// TIA Portal V17 export
// export: Created 2025-06-26T06:49:10.750176Z, ExportSetting WithDefaults, DisplayName Totally Integrated Automation Portal, DisplayVersion V17 Update 8, DisplayName TIA Portal Openness, DisplayVersion V17 Update 8, DisplayName TIA Portal Version Control Interface, DisplayVersion V17, DisplayName STEP 7 Professional, DisplayVersion V17 Update 8, DisplayName STEP 7 Safety, DisplayVersion V17 Update 6, DisplayName WinCC Advanced, DisplayVersion V17 Update 8
FUNCTION_BLOCK "DigitalInputProcessing"   // FB8, FBD
TITLE = Handle digital input signals
{ S7_Optimized_Access := 'TRUE' }
AUTHOR : Heaten
VERSION : 0.1
// Map, validate and process digital inputs
// stored: AutoNumber true, IsIECCheckEnabled false, IsRetainMemResEnabled false, MemoryReserve 0, SetENOAutomatically false, UDAEnableTagReadback false
   VAR
      HBL_LS_632 { ExternalAccessible := 'False'; ExternalVisible := 'False'; ExternalWritable := 'False'} : "stAnalogInput";
      HBL_LS_633 { S7_SetPoint := 'True'} : "stAnalogInput";
      HBL_LS_644 { S7_SetPoint := 'True'} : "stAnalogInput";
      HBL_LS_674 { S7_SetPoint := 'True'} : "stAnalogInput";
      Dummy { ExternalAccessible := 'False'; ExternalVisible := 'False'; ExternalWritable := 'False'} : Bool;
      LS632 : Real;
      LS633 : Real;
      LS644 : Real;
      LS674 : Real;
   END_VAR
   // HBL_LS_632.Raw.iMin := 0;
   // HBL_LS_632.Raw.iMax := 27648;
   // HBL_LS_632.Eng.fMin := 4.0;   // [mA]
   // HBL_LS_632.Eng.fMax := 20.0;   // [mA]
   // HBL_LS_633.Raw.iMin := 0;
   // HBL_LS_633.Raw.iMax := 27648;
   // HBL_LS_633.Eng.fMin := 4.0;   // [mA]
   // HBL_LS_633.Eng.fMax := 20.0;   // [mA]
   // HBL_LS_644.Eng.fMin := 4.0;
   // HBL_LS_644.Eng.fMax := 20.0;
   // HBL_LS_674.Eng.fMin := 4.0;
   // HBL_LS_674.Eng.fMax := 20.0;
BEGIN

REGION Network 1: Emergency stop status
   // Polarity of input is preserved. 1 = No E-stop, 0 = E-stop
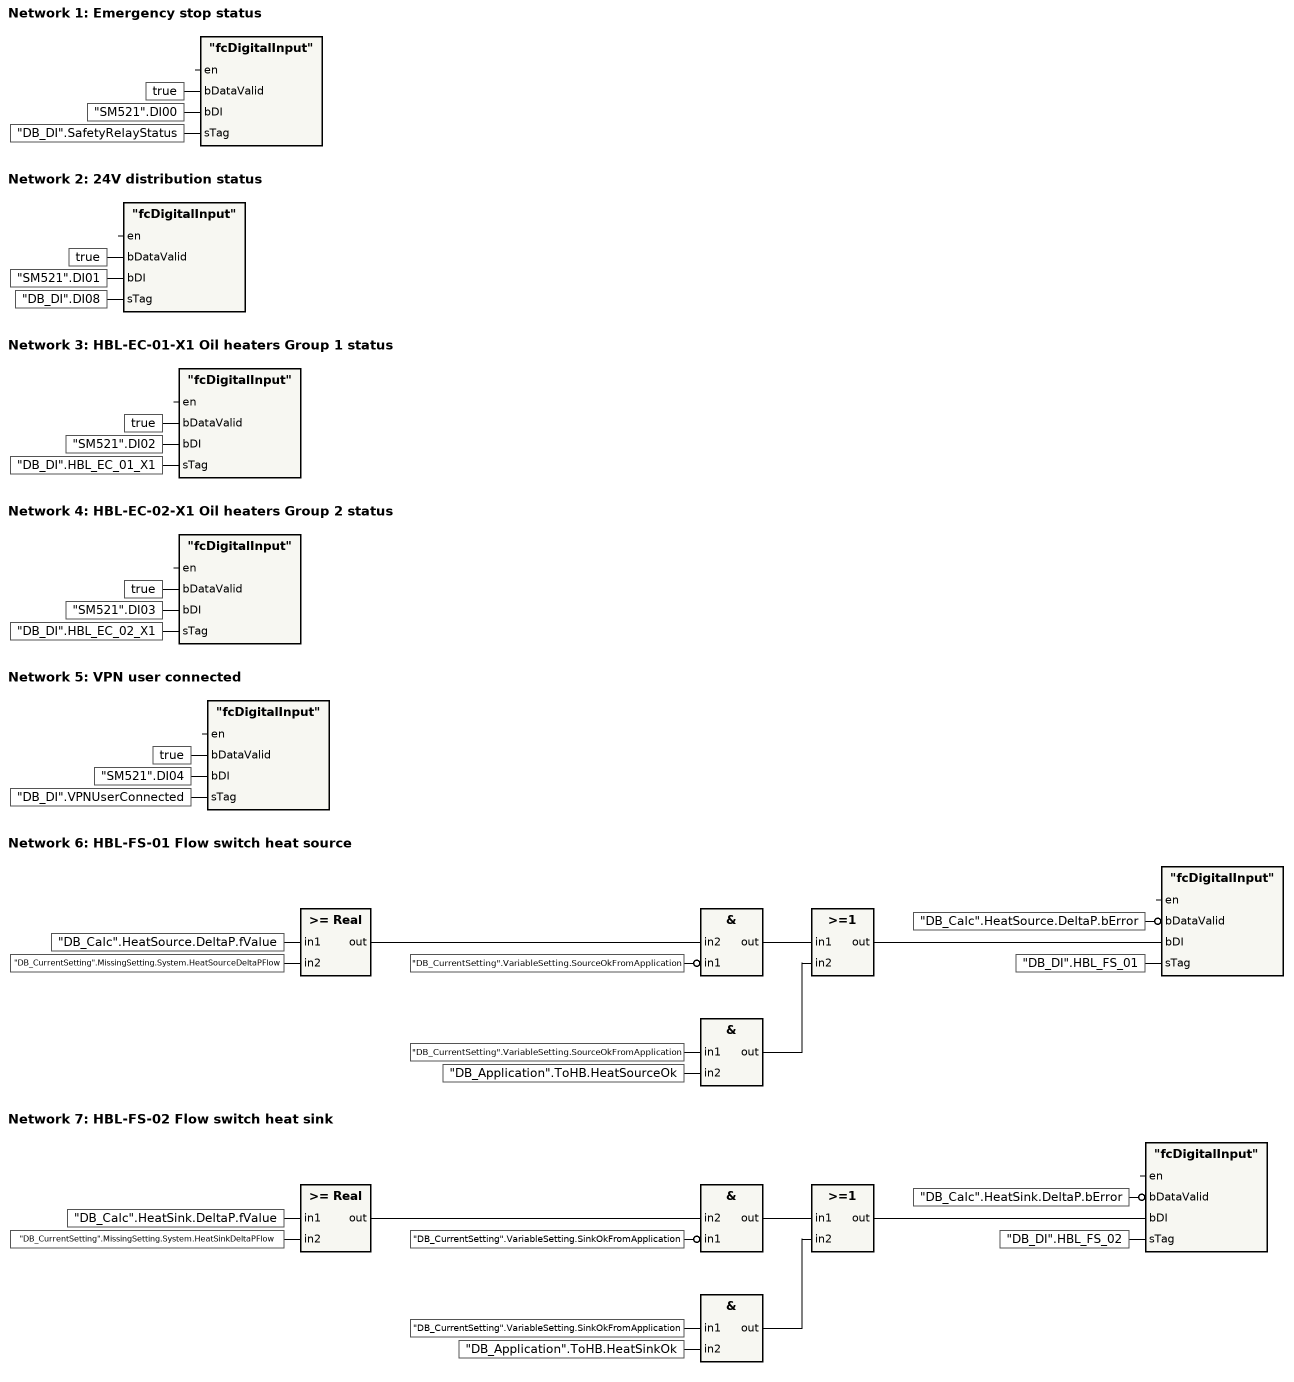
   "fcDigitalInput"(bDataValid := true, bDI := "SM521".DI00, sTag := "DB_DI".SafetyRelayStatus);
END_REGION

REGION Network 2: 24V distribution status
   "fcDigitalInput"(bDataValid := true, bDI := "SM521".DI01, sTag := "DB_DI".DI08);
END_REGION

REGION Network 3: HBL-EC-01-X1 Oil heaters Group 1 status
   "fcDigitalInput"(bDataValid := true, bDI := "SM521".DI02, sTag := "DB_DI".HBL_EC_01_X1);
END_REGION

REGION Network 4: HBL-EC-02-X1 Oil heaters Group 2 status
   "fcDigitalInput"(bDataValid := true, bDI := "SM521".DI03, sTag := "DB_DI".HBL_EC_02_X1);
END_REGION

REGION Network 5: VPN user connected
   "fcDigitalInput"(bDataValid := true, bDI := "SM521".DI04, sTag := "DB_DI".VPNUserConnected);
END_REGION

REGION Network 6: HBL-FS-01 Flow switch heat source
   // Virtual instrument:
   //  - Generate this locally from the pressure difference across the evaporator
   //  - Let the Application PLC do it based on input from the host process
   "fcDigitalInput"(bDataValid := NOT "DB_Calc".HeatSource.DeltaP.bError,
                    bDI := (("DB_Calc".HeatSource.DeltaP.fValue >= "DB_CurrentSetting".MissingSetting.System.HeatSourceDeltaPFlow) AND NOT "DB_CurrentSetting".VariableSetting.SourceOkFromApplication) OR ("DB_CurrentSetting".VariableSetting.SourceOkFromApplication AND "DB_Application".ToHB.HeatSourceOk),
                    sTag := "DB_DI".HBL_FS_01);
END_REGION

REGION Network 7: HBL-FS-02 Flow switch heat sink
   // Virtual instrument:
   //  - Generate this from the pressure difference across the condenser
   //  - Let the Application PLC does it based on input from the host process
   "fcDigitalInput"(bDataValid := NOT "DB_Calc".HeatSink.DeltaP.bError,
                    bDI := (("DB_Calc".HeatSink.DeltaP.fValue >= "DB_CurrentSetting".MissingSetting.System.HeatSinkDeltaPFlow) AND NOT "DB_CurrentSetting".VariableSetting.SinkOkFromApplication) OR ("DB_CurrentSetting".VariableSetting.SinkOkFromApplication AND "DB_Application".ToHB.HeatSinkOk),
                    sTag := "DB_DI".HBL_FS_02);
END_REGION

REGION Network 8: HBL-PS-500-X2 Compressor discharge overpressure
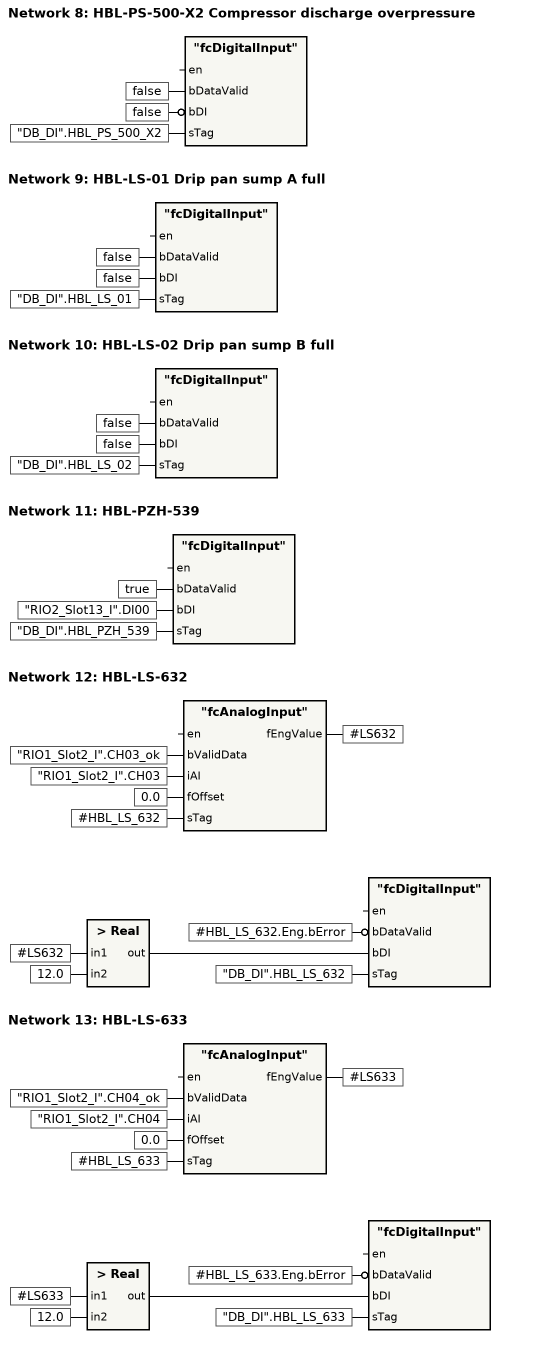
   "fcDigitalInput"(bDataValid := false, bDI := NOT false, sTag := "DB_DI".HBL_PS_500_X2);
END_REGION

REGION Network 9: HBL-LS-01 Drip pan sump A full
   "fcDigitalInput"(bDataValid := false, bDI := false, sTag := "DB_DI".HBL_LS_01);
END_REGION

REGION Network 10: HBL-LS-02 Drip pan sump B full
   "fcDigitalInput"(bDataValid := false, bDI := false, sTag := "DB_DI".HBL_LS_02);
END_REGION

REGION Network 11: HBL-PZH-539
   "fcDigitalInput"(bDataValid := true, bDI := "RIO2_Slot13_I".DI00, sTag := "DB_DI".HBL_PZH_539);
END_REGION

REGION Network 12: HBL-LS-632
   // 2-wire level switch. Low = 8mA, High = 16mA. Use a 12mA threshold to switch HI/LO
   "fcAnalogInput"(bValidData := "RIO1_Slot2_I".CH03_ok,
                   iAI := "RIO1_Slot2_I".CH03,
                   fOffset := 0.0,
                   sTag := #HBL_LS_632,
                   fEngValue => #LS632);
   "fcDigitalInput"(bDataValid := NOT #HBL_LS_632.Eng.bError, bDI := #LS632 > 12.0, sTag := "DB_DI".HBL_LS_632);
END_REGION

REGION Network 13: HBL-LS-633
   // 2-wire level switch. Low = 8mA, High = 16mA. Use a 12mA threshold to switch HI/LO
   "fcAnalogInput"(bValidData := "RIO1_Slot2_I".CH04_ok,
                   iAI := "RIO1_Slot2_I".CH04,
                   fOffset := 0.0,
                   sTag := #HBL_LS_633,
                   fEngValue => #LS633);
   "fcDigitalInput"(bDataValid := NOT #HBL_LS_633.Eng.bError, bDI := #LS633 > 12.0, sTag := "DB_DI".HBL_LS_633);
END_REGION

REGION Network 14: HBL-LS-644
   // 2-wire level switch. Low = 8mA, High = 16mA. Use a 12mA threshold to switch HI/LO
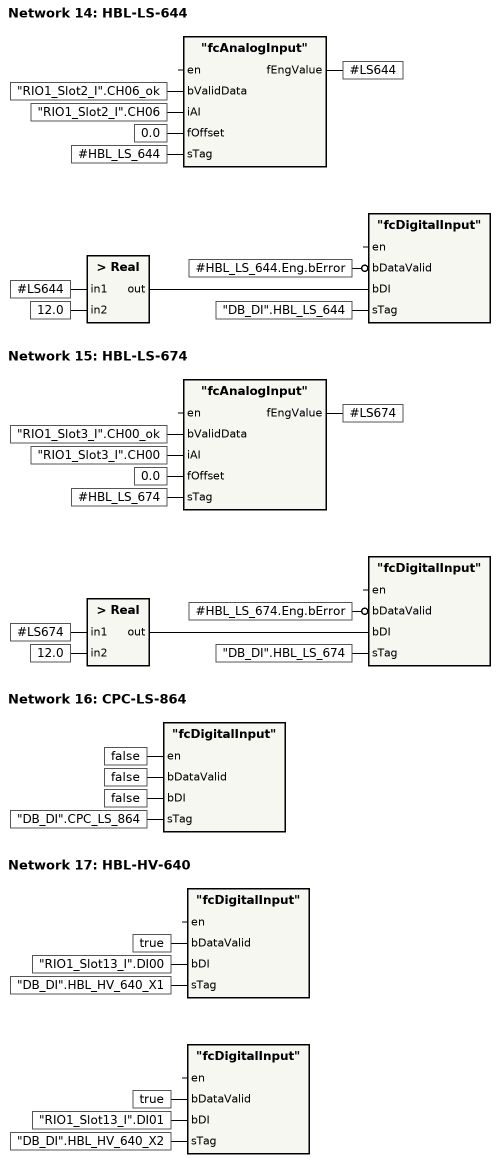
   "fcAnalogInput"(bValidData := "RIO1_Slot2_I".CH06_ok,
                   iAI := "RIO1_Slot2_I".CH06,
                   fOffset := 0.0,
                   sTag := #HBL_LS_644,
                   fEngValue => #LS644);
   "fcDigitalInput"(bDataValid := NOT #HBL_LS_644.Eng.bError, bDI := #LS644 > 12.0, sTag := "DB_DI".HBL_LS_644);
END_REGION

REGION Network 15: HBL-LS-674
   // 2-wire level switch. Low = 8mA, High = 16mA. Use a 12mA threshold to switch HI/LO
   "fcAnalogInput"(bValidData := "RIO1_Slot3_I".CH00_ok,
                   iAI := "RIO1_Slot3_I".CH00,
                   fOffset := 0.0,
                   sTag := #HBL_LS_674,
                   fEngValue => #LS674);
   "fcDigitalInput"(bDataValid := NOT #HBL_LS_674.Eng.bError, bDI := #LS674 > 12.0, sTag := "DB_DI".HBL_LS_674);
END_REGION

REGION Network 16: CPC-LS-864
   IF false THEN "fcDigitalInput"(bDataValid := false, bDI := false, sTag := "DB_DI".CPC_LS_864); END_IF;
END_REGION

REGION Network 17: HBL-HV-640
   "fcDigitalInput"(bDataValid := true, bDI := "RIO1_Slot13_I".DI00, sTag := "DB_DI".HBL_HV_640_X1);
   "fcDigitalInput"(bDataValid := true, bDI := "RIO1_Slot13_I".DI01, sTag := "DB_DI".HBL_HV_640_X2);
END_REGION

REGION Network 18: HBL-HV-670
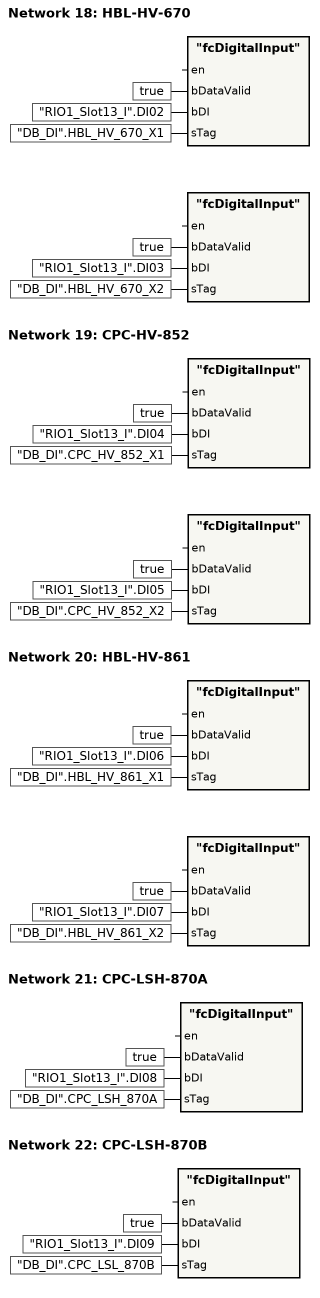
   "fcDigitalInput"(bDataValid := true, bDI := "RIO1_Slot13_I".DI02, sTag := "DB_DI".HBL_HV_670_X1);
   "fcDigitalInput"(bDataValid := true, bDI := "RIO1_Slot13_I".DI03, sTag := "DB_DI".HBL_HV_670_X2);
END_REGION

REGION Network 19: CPC-HV-852
   // '
   "fcDigitalInput"(bDataValid := true, bDI := "RIO1_Slot13_I".DI04, sTag := "DB_DI".CPC_HV_852_X1);
   "fcDigitalInput"(bDataValid := true, bDI := "RIO1_Slot13_I".DI05, sTag := "DB_DI".CPC_HV_852_X2);
END_REGION

REGION Network 20: HBL-HV-861
   // '
   "fcDigitalInput"(bDataValid := true, bDI := "RIO1_Slot13_I".DI06, sTag := "DB_DI".HBL_HV_861_X1);
   "fcDigitalInput"(bDataValid := true, bDI := "RIO1_Slot13_I".DI07, sTag := "DB_DI".HBL_HV_861_X2);
END_REGION

REGION Network 21: CPC-LSH-870A
   "fcDigitalInput"(bDataValid := true, bDI := "RIO1_Slot13_I".DI08, sTag := "DB_DI".CPC_LSH_870A);
END_REGION

REGION Network 22: CPC-LSH-870B
   "fcDigitalInput"(bDataValid := true, bDI := "RIO1_Slot13_I".DI09, sTag := "DB_DI".CPC_LSL_870B);
END_REGION

REGION Network 23: CPC-PZH-874
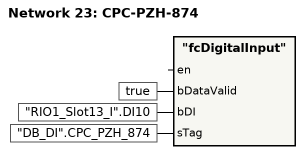
   "fcDigitalInput"(bDataValid := true, bDI := "RIO1_Slot13_I".DI10, sTag := "DB_DI".CPC_PZH_874);
END_REGION
END_FUNCTION_BLOCK
